FUNCTION TFRefreshUsedCode : BOOL
VAR_INPUT
	pcode : INT;
	UsedCode : POINTER TO ARRAY [1..MAXFORMINGCODE] OF INT;
END_VAR
VAR
	j : INT;
END_VAR

TFRefreshUsedCode := FALSE;

FOR j:=1 TO MAXFORMINGCODE-1 DO
	UsedCode^[MAXFORMINGCODE-j+1]:= UsedCode^[MAXFORMINGCODE-j];
END_FOR
UsedCode^[1] := pcode;

TFRefreshUsedCode := TRUE;

END_FUNCTION

(* stored: Version 1.1.0.1, ProductVersion 3.1.4024.11
   POU TFRefreshUsedCode: Id {e4d5b804-198b-4a3d-8af6-235ea9493b8e}, SpecialFunc None *)
